// TIA Portal V19 export
DATA_BLOCK "DB_Daten_Heraeus"   // DB1111
{ S7_Optimized_Access := 'FALSE' }
// stored: AutoNumber false
   VAR RETAIN
      "Leitwert_CM01.BN01" : Real;   // Leitfähigkeit Bypass Filterpumpe
      "Leitwert_CM01.BN02" : Real;   // Leitfähigkeit Düsen Umwälzung
      "Leitwert_CM02.BN03" : Real;   // Leitfähigkeit Bypass Filterpumpe
      "Leitwert_CM02.BN04" : Real;   // Leitfähigkeit Düsen Umwälzung
      "p_HQ01.BP01" : Real;   // Druck Beutelfiltergehäuse
      "p_HQ02.BP02" : Real;   // Druck Beutelfiltergehäuse
      "p_CM01.BP03" : Real;   // Druck Filterpumpe
      "p_CM01.BP04" : Real;   // Druck Umwälzpumpe
      "p_CM03.BP05" : Real;   // Druck Umwäzpumpe
      "p_CM02.BP06" : Real;   // Druck Filterpumpe
      "p_CM02.BP07" : Real;   // Druck Umwälzpumpe
      "p_CM04.BP08" : Real;   // Druck Umwäzpumpe
      "p_CM05.BP09" : Real;   // Druck Pumpe Entleerung Sammeltank
   END_VAR
BEGIN
END_DATA_BLOCK
